(* IEC 61131-3 sources: CtrlxLadderSkill/references/examples, 3 files *)

(* ---- E_CycleState.st ---- *)
{attribute 'qualified_only'}
{attribute 'strict'}
TYPE E_CycleState :
(
    Idle := 0,
    Clamping,
    Working,
    Unclamping,
    Done,
    Aborting,
    Faulted
) UINT;
END_TYPE

(* ---- FB_AxisCtrl.st ---- *)
// FB_AxisCtrl in ladder, from the PressSystem project (2026-10-10). Schema-valid and scan-tested in ld_sim with
// fake MC_ models (press_tests/test_axisctrl.py); NOT yet compiled in ctrlX PLC Engineering.
// FB_AxisCtrl: one ctrlX axis through CXA_PLCopen: power, absolute move, halt, reset and status.
// Latches the first error with its ctrlX diagnosis until reset. Not a sequence; the caller drives it.
FUNCTION_BLOCK FB_AxisCtrl
VAR_INPUT
    bPower          : BOOL;         // power on (level)
    bMove           : BOOL;         // absolute move (Execute): needs a FALSE->TRUE edge per move
    lrPosition      : LREAL;        // absolute target, taken at the edge of bMove
    stDyn           : ST_Dynamics;  // move dynamics, taken at the edge of bMove
    bHalt           : BOOL;         // halt (Execute, level)
    lrHaltDec       : LREAL;        // halt deceleration
    bReset          : BOOL;         // reset latched error and drive ErrorStop (level)
END_VAR
VAR_OUTPUT
    bPowered        : BOOL;         // power on and confirmed
    bStandstill     : BOOL;         // powered, not moving, no error
    bInPos          : BOOL;         // current move done (held while bMove is TRUE)
    bHalted         : BOOL;         // halt done (held while bHalt is TRUE)
    bError          : BOOL;         // latched error (FB error or axis ErrorStop)
    lrActPos        : LREAL;        // actual position (valid while powered)
    eErrorID        : ERROR_CODE;   // latched error class
    dwDiagMain      : DWORD;        // latched ctrlX main diagnosis (0 for a drive ErrorStop: see ctrlX diagnostics)
    dwDiagDetail    : DWORD;        // latched ctrlX detail diagnosis
END_VAR
VAR_IN_OUT
    stAxis          : AXIS_REF;     // axis to control
END_VAR
VAR
    _bError         : BOOL;
    _eErrorID       : ERROR_CODE;
    _dwDiagMain     : DWORD;
    _dwDiagDetail   : DWORD;
    _bPowerEnable   : BOOL;         // MC_Power.Enable
    _bStatusEnable  : BOOL;         // MC_ReadStatus.Enable
    _bActPosEnable  : BOOL;         // MC_ReadActualPosition.Enable
    _bResetExecute  : BOOL;         // MC_Reset.Execute
    _bMoveExecute   : BOOL;         // MC_MoveAbsolute.Execute
    _bHaltExecute   : BOOL;         // MC_Halt.Execute
    _fbPower        : MC_Power;
    _fbReset        : MC_Reset;
    _fbStatus       : MC_ReadStatus;
    _fbActPos       : MC_ReadActualPosition;
    _fbMove         : MC_MoveAbsolute;
    _fbHalt         : MC_Halt;
END_VAR

// ===== Error latch: sub-FB results are from the previous scan, the same as a timer's Q =====
NETWORK Clear error
// Reset clears the latch once the drive has left ErrorStop
    _bError bReset /_fbStatus.ErrorStop /_fbReset.Active
        -> R:_bError, _eErrorID := ERROR_CODE.NONE_ERROR, _dwDiagMain := 0, _dwDiagDetail := 0

NETWORK Latch MC_Power error
// Each latch rung sets _bError, which locks out the rungs below: the first error is kept
    /_bError _fbPower.Error
        -> S:_bError, _eErrorID := _fbPower.ErrorID,
           _dwDiagMain := _fbPower.ErrorIdent.Additional1, _dwDiagDetail := _fbPower.ErrorIdent.Additional2

NETWORK Latch MC_MoveAbsolute error
    /_bError _fbMove.Error
        -> S:_bError, _eErrorID := _fbMove.ErrorID,
           _dwDiagMain := _fbMove.ErrorIdent.Additional1, _dwDiagDetail := _fbMove.ErrorIdent.Additional2

NETWORK Latch MC_Halt error
    /_bError _fbHalt.Error
        -> S:_bError, _eErrorID := _fbHalt.ErrorID,
           _dwDiagMain := _fbHalt.ErrorIdent.Additional1, _dwDiagDetail := _fbHalt.ErrorIdent.Additional2

NETWORK Latch MC_Reset error
    /_bError _fbReset.Error
        -> S:_bError, _eErrorID := _fbReset.ErrorID,
           _dwDiagMain := _fbReset.ErrorIdent.Additional1, _dwDiagDetail := _fbReset.ErrorIdent.Additional2

NETWORK Latch MC_ReadStatus error
    /_bError _fbStatus.Error
        -> S:_bError, _eErrorID := _fbStatus.ErrorID,
           _dwDiagMain := _fbStatus.ErrorIdent.Additional1, _dwDiagDetail := _fbStatus.ErrorIdent.Additional2

NETWORK Latch axis ErrorStop
// Error raised in the drive/motion kernel while moving; the detail is in the ctrlX diagnostics log
    /_bError _fbStatus.Valid _fbStatus.ErrorStop
        -> S:_bError, _eErrorID := ERROR_CODE.DEVICE_ERROR, _dwDiagMain := 0, _dwDiagDetail := 0

// ===== FB inputs =====
NETWORK MC_Power enable
// A failed Power (e.g. motion not RUNNING yet) needs a new edge: reset drops Enable for one scan
    bPower (/_fbPower.Error | /bReset) -> _bPowerEnable

NETWORK MC_ReadStatus enable
// Read only while powered, so a switched-off system doesn't fault at boot
    bPower (/_fbStatus.Error | /bReset) -> _bStatusEnable

NETWORK MC_ReadActualPosition enable
    bPower (/_fbActPos.Error | /bReset) -> _bActPosEnable

NETWORK MC_Reset execute
    bReset _fbStatus.ErrorStop -> _bResetExecute

NETWORK MC_MoveAbsolute execute
    bMove /_bError -> _bMoveExecute

NETWORK MC_Halt execute
// No halt on an unpowered axis or one in ErrorStop: the drive has already stopped it
    bHalt _fbPower.Status /_fbStatus.ErrorStop -> _bHaltExecute

// ===== Sub-FBs, every scan =====
NETWORK Power
    -> _fbPower(Enable := _bPowerEnable, Axis := stAxis)

NETWORK Read status
    -> _fbStatus(Enable := _bStatusEnable, Axis := stAxis)

NETWORK Read actual position
    -> _fbActPos(Enable := _bActPosEnable, Axis := stAxis)

NETWORK Reset
    -> _fbReset(Execute := _bResetExecute, Axis := stAxis)

NETWORK Move absolute
    -> _fbMove(Execute := _bMoveExecute, Position := lrPosition, Velocity := stDyn.lrVel,
               Acceleration := stDyn.lrAcc, Deceleration := stDyn.lrDec, Jerk := stDyn.lrJerk,
               BufferMode := MC_BUFFER_MODE.mcAborting, Axis := stAxis)

NETWORK Halt
// The manual's interface table calls the axis pin 'Axes'; rename here if the compiler rejects 'Axis'
    -> _fbHalt(Execute := _bHaltExecute, Deceleration := lrHaltDec, Jerk := 0.0, Axis := stAxis)

// ===== Outputs, last =====
NETWORK Out bPowered
    _fbPower.Status -> bPowered

NETWORK Out bStandstill
    _fbStatus.Valid _fbStatus.Standstill -> bStandstill

NETWORK Out bInPos
// Gated by the command so a Done can never outlive the step that asked for it
    _fbMove.Done bMove -> bInPos

NETWORK Out bHalted
    _fbHalt.Done bHalt -> bHalted

NETWORK Out bError
    _bError -> bError

NETWORK Out copies
    -> lrActPos := _fbActPos.Position, eErrorID := _eErrorID,
       dwDiagMain := _dwDiagMain, dwDiagDetail := _dwDiagDetail
END_FUNCTION_BLOCK

(* ---- FB_CycleLD.st ---- *)
// FB_CycleLD: one clamp/work/unclamp cycle per Execute, with abort, step timeouts and latched faults.
// Ladder version of FB_Cycle: jumps -> commit -> transitions -> commit -> state decode -> on change
// -> FB calls -> outputs. After the decode the logic uses contacts, never compares in parallel.
FUNCTION_BLOCK FB_CycleLD
VAR_INPUT
    bExecute        : BOOL;     // run one cycle; hold TRUE until Done/Error, then remove
    bAbort          : BOOL;     // abort request (level), e.g. guard opened
    bReset          : BOOL;     // fault reset (level), only acts once Execute is removed
    bExternalFault  : BOOL;     // fault cause from outside, e.g. drive fault
    bClamped        : BOOL;     // feedback: clamp closed
    bUnclamped      : BOOL;     // feedback: clamp open
    bWorkDone       : BOOL;     // feedback: work station finished
END_VAR
VAR_OUTPUT
    eState          : E_CycleState; // current step, for HMI / online view
    bBusy           : BOOL;         // cycle in progress
    bDone           : BOOL;         // cycle finished; held until Execute is removed
    bError          : BOOL;         // faulted; held until reset with Execute removed
    uiFaultCode     : UINT;         // first fault that latched, 0 = none
    eFaultState     : E_CycleState; // step that was active when the fault latched
    bClampCmd       : BOOL;         // valve: close clamp
    bWorkCmd        : BOOL;         // start work station
END_VAR
VAR
    _eState         : E_CycleState; // the state; eState is only a copy for the caller
    _eNextState     : E_CycleState; // written by jumps/transitions, committed to _eState after each section
    _eLastState     : E_CycleState;
    _bStateChanged  : BOOL;         // TRUE on the scan the state changed (on-change section)
    _uiFaultCode    : UINT;
    _eFaultState    : E_CycleState;
    _tStepTimeout   : TIME;         // timeout of the current step, T#0S = none
    _bStIdle        : BOOL;         // state decoded after the commit: one BOOL per state
    _bStClamping    : BOOL;
    _bStWorking     : BOOL;
    _bStUnclamping  : BOOL;
    _bStDone        : BOOL;
    _bStAborting    : BOOL;
    _bStFaulted     : BOOL;
    _fbStepTimer    : TON;
END_VAR
VAR CONSTANT
    CLAMP_TIMEOUT       : TIME := T#3S;
    WORK_TIMEOUT        : TIME := T#30S;
    UNCLAMP_TIMEOUT     : TIME := T#3S;
    FAULT_NONE          : UINT := 0;
    FAULT_EXTERNAL      : UINT := 1;
    FAULT_STEP_TIMEOUT  : UINT := 2;
    FAULT_INVALID_STATE : UINT := 99;
END_VAR

// ===== 1. Jumps: highest priority first, each one locks out the ones below =====
NETWORK J1 External fault
    [_eState <> E_CycleState.Faulted] bExternalFault
        -> _eNextState := E_CycleState.Faulted, _uiFaultCode := FAULT_EXTERNAL, _eFaultState := _eState

NETWORK J2 Step timeout
// The step timer belongs to the current step, so this one rung covers every step's timeout
    [_eState <> E_CycleState.Faulted] /bExternalFault _fbStepTimer.Q
        -> _eNextState := E_CycleState.Faulted, _uiFaultCode := FAULT_STEP_TIMEOUT, _eFaultState := _eState

NETWORK J3 Abort while clamping
// One compare per rung: abort in two states is two networks (neither state is Faulted)
    [_eState = E_CycleState.Clamping] /bExternalFault /_fbStepTimer.Q bAbort
        -> _eNextState := E_CycleState.Aborting

NETWORK J4 Abort while working
    [_eState = E_CycleState.Working] /bExternalFault /_fbStepTimer.Q bAbort
        -> _eNextState := E_CycleState.Aborting

NETWORK Commit jumps
    -> _eState := _eNextState

// ===== 2. Transitions only =====
NETWORK T Idle -> Clamping
    [_eState = E_CycleState.Idle] bExecute /bAbort -> _eNextState := E_CycleState.Clamping

NETWORK T Clamping -> Working
    [_eState = E_CycleState.Clamping] bClamped -> _eNextState := E_CycleState.Working

NETWORK T Working -> Unclamping
    [_eState = E_CycleState.Working] bWorkDone -> _eNextState := E_CycleState.Unclamping

NETWORK T Unclamping -> Done
    [_eState = E_CycleState.Unclamping] bUnclamped -> _eNextState := E_CycleState.Done

NETWORK T Done -> Idle
// Hold until the command is removed: this is what replaces an edge on Execute
    [_eState = E_CycleState.Done] /bExecute -> _eNextState := E_CycleState.Idle

NETWORK T Aborting -> Idle
    [_eState = E_CycleState.Aborting] bUnclamped /bExecute -> _eNextState := E_CycleState.Idle

NETWORK T Faulted -> Idle
    [_eState = E_CycleState.Faulted] bReset /bExecute /bExternalFault -> _eNextState := E_CycleState.Idle

NETWORK T Invalid state -> Faulted
// The CASE ELSE: any value past the last state (e.g. after an online change)
    [_eState > E_CycleState.Faulted]
        -> _eNextState := E_CycleState.Faulted, _uiFaultCode := FAULT_INVALID_STATE, _eFaultState := _eState

NETWORK Commit transitions
    -> _eState := _eNextState

// ===== State decode: one compare per rung, so later rungs use contacts =====
NETWORK Decode Idle
    [_eState = E_CycleState.Idle] -> _bStIdle

NETWORK Decode Clamping
    [_eState = E_CycleState.Clamping] -> _bStClamping

NETWORK Decode Working
    [_eState = E_CycleState.Working] -> _bStWorking

NETWORK Decode Unclamping
    [_eState = E_CycleState.Unclamping] -> _bStUnclamping

NETWORK Decode Done
    [_eState = E_CycleState.Done] -> _bStDone

NETWORK Decode Aborting
    [_eState = E_CycleState.Aborting] -> _bStAborting

NETWORK Decode Faulted
    [_eState = E_CycleState.Faulted] -> _bStFaulted

// ===== 3. On change: common actions, then entry actions of the new state =====
NETWORK State changed
    [_eState <> _eLastState] -> _bStateChanged

NETWORK Common: no timeout unless the new step sets one
    _bStateChanged -> _tStepTimeout := T#0S

NETWORK Entry Idle
// Idle means no fault: fault info only exists while the sequence is out of Idle
    _bStateChanged _bStIdle -> _uiFaultCode := FAULT_NONE, _eFaultState := E_CycleState.Idle

NETWORK Entry Clamping
    _bStateChanged _bStClamping -> _tStepTimeout := CLAMP_TIMEOUT

NETWORK Entry Working
    _bStateChanged _bStWorking -> _tStepTimeout := WORK_TIMEOUT

NETWORK Entry Unclamping, Aborting
    _bStateChanged (_bStUnclamping | _bStAborting) -> _tStepTimeout := UNCLAMP_TIMEOUT

NETWORK Remember state
    -> _eLastState := _eState

// ===== 4. Cyclic: every sub-FB call, then every output last =====
NETWORK Step timer
// Off for the change scan, so it restarts in every new step
    [_tStepTimeout > T#0S] /_bStateChanged _fbStepTimer(PT := _tStepTimeout)

NETWORK Out bBusy
    (_bStClamping | _bStWorking | _bStUnclamping | _bStAborting) -> bBusy

NETWORK Out bDone
    _bStDone -> bDone

NETWORK Out bError
    _bStFaulted -> bError

NETWORK Out bClampCmd
// Aborting opens the clamp
    (_bStClamping | _bStWorking) -> bClampCmd

NETWORK Out bWorkCmd
    _bStWorking -> bWorkCmd

NETWORK Out copies
// The logic above never reads its own outputs
    -> eState := _eState, uiFaultCode := _uiFaultCode, eFaultState := _eFaultState
END_FUNCTION_BLOCK
